// TIA Portal V17 export
// export: Created 2026-04-13T11:12:45.095747Z, ExportSetting WithDefaults, DisplayName Totally Integrated Automation Portal, DisplayVersion V17 Update 4, DisplayName TIA Portal Openness, DisplayVersion V17 Update 4, DisplayName TIA Portal Version Control Interface, DisplayVersion V17, DisplayName SINAMICS Startdrive Advanced, DisplayVersion V17, DisplayName SINAMICS Startdrive G130, G150, S120, S150, SINAMICS MV, S210, DisplayVersion V17, DisplayName SINAMICS Startdrive G110M, G120, G120C, G120D, G120P, G115D, DisplayVersion V17, DisplayName STEP 7 Professional, DisplayVersion V17 Update 4, DisplayName STEP 7 Safety, DisplayVersion V17, DisplayName WinCC Professional, DisplayVersion V17 Update 4
VAR_GLOBAL   // PLC tag table "AIQ"
   IW100 AT %IW100 : Int;
   IW102 AT %IW102 : Int;
   IW104 AT %IW104 : Int;
   IW106 AT %IW106 : Int;
   IW108 AT %IW108 : Int;
   IW110 AT %IW110 : Int;
   IW112 AT %IW112 : Int;
   IW116 AT %IW116 : Int;
   IW118 AT %IW118 : Int;
   IW120 AT %IW120 : Int;
   IW122 AT %IW122 : Int;
   IW124 AT %IW124 : Int;
   IW126 AT %IW126 : Int;
   IW128 AT %IW128 : Int;
   IW130 AT %IW130 : Int;
   IW132 AT %IW132 : Int;
   IW134 AT %IW134 : Int;
   IW136 AT %IW136 : Int;
   IW138 AT %IW138 : Int;
   IW140 AT %IW140 : Int;
   IW142 AT %IW142 : Int;
   QW100 AT %QW100 : Int;
   QW102 AT %QW102 : Int;
   QW104 AT %QW104 : Int;
   QW106 AT %QW106 : Int;
   QW108 AT %QW108 : Int;
   QW110 AT %QW110 : Int;
   QW112 AT %QW112 : Int;
   QW114 AT %QW114 : Int;
   QW116 AT %QW116 : Int;
   QW118 AT %QW118 : Int;
   QW120 AT %QW120 : Int;
   QW122 AT %QW122 : Int;
   QW124 AT %QW124 : Int;
   QW126 AT %QW126 : Int;
   QW128 AT %QW128 : Int;
   QW130 AT %QW130 : Int;
   QW132 AT %QW132 : Int;
   QW134 AT %QW134 : Int;
   QW136 AT %QW136 : Int;
   QW138 AT %QW138 : Int;
   QW140 AT %QW140 : Int;
   QW142 AT %QW142 : Int;
   QW144 AT %QW144 : Int;
   QW146 AT %QW146 : Int;
   QW148 AT %QW148 : Int;
   QW150 AT %QW150 : Int;
   IW114 AT %IW114 : Int;
   IW144 AT %IW144 : Int;
   IW146 AT %IW146 : Int;
   IW148 AT %IW148 : Int;
   IW150 AT %IW150 : Int;
   IW152 AT %IW152 : Int;
   IW154 AT %IW154 : Int;
   IW156 AT %IW156 : Int;
   IW158 AT %IW158 : Int;
   IW160 AT %IW160 : Int;
   IW162 AT %IW162 : Int;
END_VAR
